FUNCTION_BLOCK Bohrkopf
VAR_INPUT
END_VAR
VAR_OUTPUT
	Done: BOOL := FALSE;
	Stopped: BOOL := TRUE;
	Initialized: BOOL := FALSE;
END_VAR
VAR
	axisRef: AXIS_REF;
	fbMcMove: MC_MoveAbsolute;
	fbMcPower: MC_Power;
	fbMcStop: MC_Stop;
	eZustand: E_STATES_BOHRKOPF := E_STATES_BOHRKOPF.stopped;
	
	stConfig: REFERENCE TO ST_Config;
	
	// Stop-Command set via outside call?
	bDoStop: BOOL := FALSE;
END_VAR

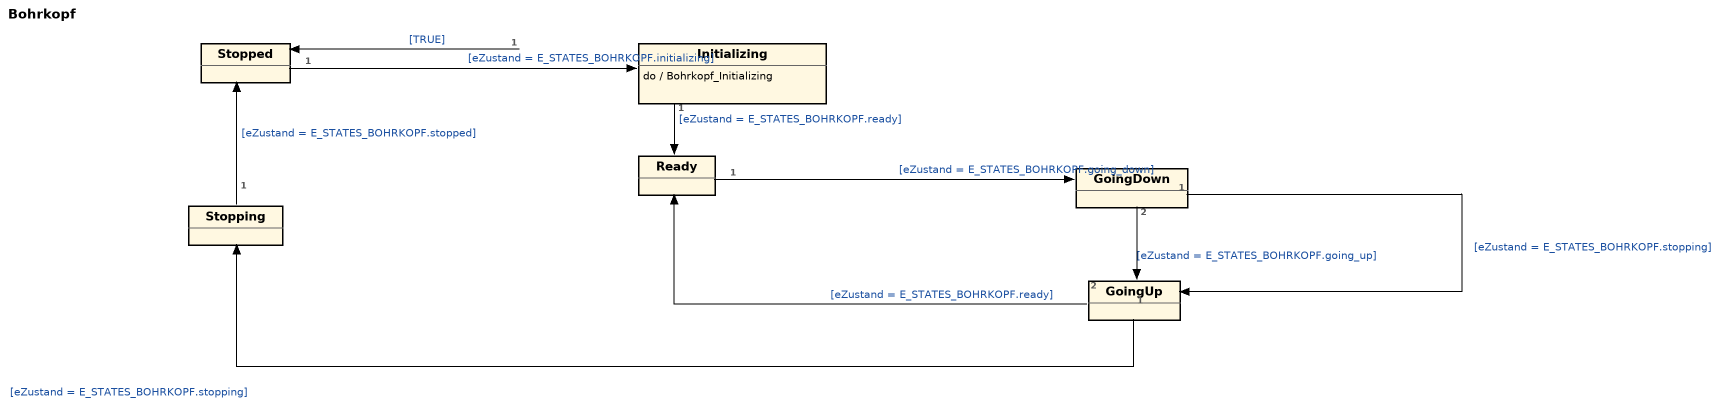
STATECHART Bohrkopf  // abortable
    START StartState1
    STATE Stopped
    STATE Initializing
        do / Bohrkopf_Initializing
    STATE Ready
    STATE GoingDown
    STATE Stopping
    STATE GoingUp
    StartState1 -> Stopped [TRUE] // priority 1, on completion
    Stopped -> Initializing [eZustand = E_STATES_BOHRKOPF.initializing] // priority 1
    Initializing -> Ready [eZustand = E_STATES_BOHRKOPF.ready] // priority 1
    Ready -> GoingDown [eZustand = E_STATES_BOHRKOPF.going_down] // priority 1
    GoingDown -> GoingUp [eZustand = E_STATES_BOHRKOPF.stopping] // priority 1
    GoingDown -> GoingUp [eZustand = E_STATES_BOHRKOPF.going_up] // priority 2
    Stopping -> Stopped [eZustand = E_STATES_BOHRKOPF.stopped] // priority 1
    GoingUp -> Stopping [eZustand = E_STATES_BOHRKOPF.stopping] // priority 1
    GoingUp -> Ready [eZustand = E_STATES_BOHRKOPF.ready] // priority 2
END_STATECHART

METHOD PUBLIC Bohren : HRESULT
VAR_INPUT
END_VAR
CASE eZustand OF
	E_STATES_BOHRKOPF.ready:
		// bohren starten
		eZustand := E_STATES_BOHRKOPF.going_down;
		Bohren := S_PENDING;
		
	ELSE
		// bohrend
		Bohren := S_PENDING;
END_CASE
END_METHOD

METHOD Bohrkopf_Initializing : HRESULT
VAR_INPUT
END_VAR
axisRef.ReadStatus();

fbMcPower(
	Axis := axisRef,
	Enable := TRUE,
	Enable_Positive := TRUE,
	Enable_Negative := TRUE
);

IF fbMcPower.Status THEN
	THIS^.Initialized := TRUE;
	THIS^.eZustand := E_STATES_BOHRKOPF.ready;
END_IF
END_METHOD

PROPERTY PUBLIC Config : REFERENCE TO ST_Config
SET
THIS^.stConfig := Config;
END_SET
END_PROPERTY

METHOD PUBLIC GoUp : BOOL
VAR_INPUT
END_VAR
VAR_OUTPUT
	Done: BOOL := FALSE;
END_VAR
// Bohrkopf in Ausgangsposition hochfahren
END_METHOD

PROPERTY PUBLIC Ready : BOOL
GET
Ready := THIS^.eZustand = E_STATES_BOHRKOPF.ready;
END_GET
END_PROPERTY

METHOD PUBLIC Stop : BOOL
VAR_INPUT
END_VAR
//CASE eZustand OF
//	E_STATES_BOHRKOPF.ready:
//		Stop := TRUE;
		
//	ELSE
//		Stop := FALSE;
//END_CASE
END_METHOD

END_FUNCTION_BLOCK

(* stored: Version 1.1.0.1, ProductVersion 3.1.4024.3
   POU Bohrkopf: Id {19f3ca2f-0f27-4ca2-9147-8b8deadda0f9}, SpecialFunc None
   Method Bohren: Id {8ea0bb1e-96ee-44db-a489-8c4ede5e2c82}
   Method Bohrkopf_Initializing: Id {b66a3239-347a-44fb-82d1-6204197ad550}
   Property Config: Id {cdf16ded-9c53-4920-bd19-37562fc5d192}
   Set Set: Id {b8256098-d749-47f5-a578-01fdccddf1ca}
   Method GoUp: Id {24ed18d8-0e8a-45b1-8369-3a45d07eb697}
   Property Ready: Id {798c9ef3-7b89-433a-bb30-d574c998a112}
   Get Get: Id {dcc1ff8d-2b00-4a8a-b7de-bee0d3837800}
   Method Stop: Id {14c05551-3aed-4025-b559-2749c5354fd1} *)
